// TIA Portal V19 export
FUNCTION_BLOCK "TYPIC_C701_IF_KOKR"   // FB101, FBD
TITLE = TYPIC_C701_IF_KOKR: Koelkring
{ S7_Optimized_Access := 'TRUE' }
AUTHOR : OCOTECH
FAMILY : Typical
NAME : C701.712
// Logisch Object Besturing: C701.712
// 
// De interne functie Koelkring verzorgt de interne besturing, bewaking en fysieke aansturing van een kring van de collector behorend tot de klimaatinstallatie.
// Er wordt een vrijgave aan de pompen gegeven als er een koelvraag is. De drukregeling gebeurt door de pomp zelf. Antioblokkeer beveiliging is ook instelbaar op de pomp zelf.
// Indien er een tweede pomp is, wordt deze afwisselend gebruikt. Of wordt er gewisseld bij een storing van de actieve pomp.
// De collector koelkring bestaat uit 2 kringen:
//  Kring ventiloconvectoren en klimaatkasten
//  Kring koelbatterij luchtgroep
// stored: MemoryReserve 10, SetENOAutomatically false
   VAR_INPUT
      STU_IF_KOKR { ExternalAccessible := 'False'; ExternalVisible := 'False'; ExternalWritable := 'False'} : Bool;   // Sturing van de interne functie klimaatregeling (IF), koudevraag voor kring
      IN_AAN_PMP1 { ExternalAccessible := 'False'; ExternalVisible := 'False'; ExternalWritable := 'False'} : Bool;   // Terugmelding aansturing pomp 1 (1 = Aan)
      IN_AAN_PMP2 { ExternalAccessible := 'False'; ExternalVisible := 'False'; ExternalWritable := 'False'} : Bool;   // Terugmelding aansturing pomp 2 (1 = Aan)
      IN_THM_PMP1 { ExternalAccessible := 'False'; ExternalVisible := 'False'; ExternalWritable := 'False'} : Bool;   // Status thermische beveiliging (1 = OK) pomp 1
      IN_THM_PMP2 { ExternalAccessible := 'False'; ExternalVisible := 'False'; ExternalWritable := 'False'} : Bool;   // Status thermische beveiliging (1 = OK) pomp 2
      IN_DME { ExternalAccessible := 'False'; ExternalVisible := 'False'; ExternalWritable := 'False'} : Real;   // Drukmeting
      IN_TME_IN { ExternalAccessible := 'False'; ExternalVisible := 'False'; ExternalWritable := 'False'} : Real;   // Temperatuur vertrek
      IN_TME_UIT { ExternalAccessible := 'False'; ExternalVisible := 'False'; ExternalWritable := 'False'} : Real;   // Temperatuur retour
      CFG_TYD_FB { ExternalAccessible := 'False'; ExternalVisible := 'False'; ExternalWritable := 'False'} : Time;   // Vertragingstijd storing foute terugmelding
      CFG_PMP { ExternalAccessible := 'False'; ExternalVisible := 'False'; ExternalWritable := 'False'} : Bool;   // True = Kring met 2 pompen
      CFG_PMP_TYD { ExternalAccessible := 'False'; ExternalVisible := 'False'; ExternalWritable := 'False'} : Time;   // Maximale draaitijd voor wisselen pomp
   END_VAR
   VAR_OUTPUT
      VAR_IF_KOKR { ExternalAccessible := 'False'; ExternalVisible := 'False'; ExternalWritable := 'False'} : "C701_VAR_IF_KOKR_TYPIC";   // Struct met alle variabelen naar bovenliggende functies
      OUT_VGV_PMP1 { ExternalAccessible := 'False'; ExternalVisible := 'False'; ExternalWritable := 'False'} : Bool;   // Vrijgave pomp 1
      OUT_VGV_PMP2 { ExternalAccessible := 'False'; ExternalVisible := 'False'; ExternalWritable := 'False'} : Bool;   // Vrijgave pomp 2
   END_VAR
   VAR_IN_OUT
      STU_VGV_KOKR_AAN : Bool;   // Vrijgave inschakelen NIET NODIG?
   END_VAR
   VAR
      STO { ExternalWritable := 'False'} : Struct   // Storingen
         A001 : Bool;   // Storing van de motorbeveiliging van pomp 1
         A002 : Bool;   // Storing van de motorbeveiliging van pomp 2
         A003 : Bool;   // Fout temperatuurmeting vertrek
         A004 : Bool;   // Fout temperatuurmeting retour
         A005 : Bool;   // Fout drukmeting
      END_STRUCT;
      VAR { ExternalWritable := 'False'} : Struct   // Variabelen
         TME_IN : Real;   // Temperatuur vertrek
         TME_UIT : Real;   // Temperatuur retour
         DME : Real;   // Druk vertrek
         VGV_P1 : Bool;   // Vrijgave voor pomp 1
         VGV_P2 : Bool;   // Vrijgave voor pomp 2
         TYD_TOT_AAN_P1 : LInt;   // Totaal aantal draaiuren (in seconden)
         TYD_TOT_AAN_UUR_P1 : LInt;   // Totaal aantal draaiuren (in uren)
         TYD_TOT_AAN_P2 : LInt;   // Totaal aantal draaiuren (in seconden)
         TYD_TOT_AAN_UUR_P2 : LInt;   // Totaal aantal draaiuren (in uren)
         TYD_AAN_P1 : LInt;   // Aantal seconden dat pomp aangeschakeld is
         TYD_AAN_P2 : LInt;   // Aantal seconden dat pomp aangeschakeld is
      END_STRUCT;
   END_VAR
BEGIN

REGION Network 1: START
END_REGION

REGION Network 2: +++ Metingen +++
   // inlezen van vertrek- en retourtemperatuur.
END_REGION

REGION Network 3: +++ Storingen en meldingen +++
   // aanmaken van storingen en meldingen.
END_REGION

REGION Network 4: Storing A001: Storing van de motorbeveiliging van pomp 1
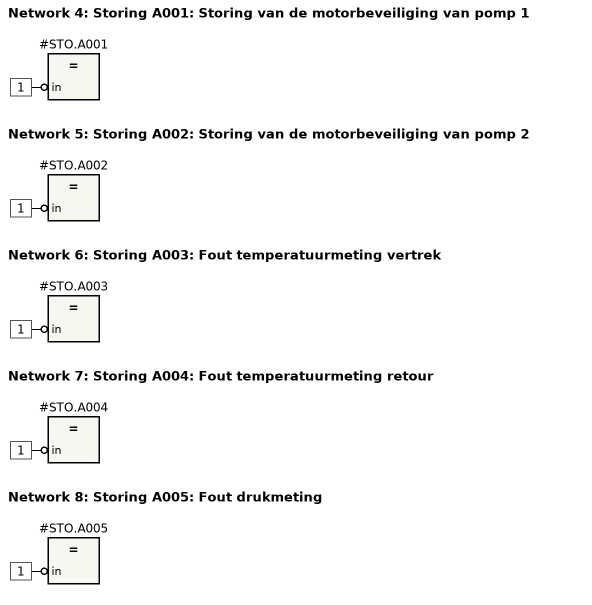
   #STO.A001 := NOT 1;
END_REGION

REGION Network 5: Storing A002: Storing van de motorbeveiliging van pomp 2
   #STO.A002 := NOT 1;
END_REGION

REGION Network 6: Storing A003: Fout temperatuurmeting vertrek
   #STO.A003 := NOT 1;
END_REGION

REGION Network 7: Storing A004: Fout temperatuurmeting retour
   #STO.A004 := NOT 1;
END_REGION

REGION Network 8: Storing A005: Fout drukmeting
   #STO.A005 := NOT 1;
END_REGION

REGION Network 9: +++ Sturingen pomp +++
   // bij koudevraag pomp vrijgave geven.
END_REGION

REGION Network 10: +++ Urentellers +++
   // tellen van de tijdsduur dat de motor draait.
END_REGION

REGION Network 11 (SCL): EINDE
   // Variabelen van intern scada rakvlak naar outputs copieren
   #VAR_IF_KOKR.STO := #STO;
END_REGION
END_FUNCTION_BLOCK
